FUNCTION_BLOCK FB_Symulacja IMPLEMENTS ITF_StanMaszyny
VAR_INPUT
	stParametry								: DUT_Symulacja_Parametry;
	stStanyPodzespolow						: DUT_Krajalnica_StanyPodzespolow;
	eTrybPracy								: E_PMLUnitMode;
END_VAR
VAR_OUTPUT
	//wyjscia zadziałania czujnikow 
	bCiecie1_Poczatek						: BOOL;
	bCiecie1_Koniec							: BOOL;
	bCiecie2_Poczatek						: BOOL;
	bCiecie2_Koniec							: BOOL;
	bPodawanieZabierakPoczatek				: BOOL;
	bPodawanieZabierakKoniec				: BOOL;
	bPodawaniePrzesuwaniePoczatek			: BOOL;
	bPodawaniePrzesuwanieKoniec				: BOOL;
	bCzujnikWaflaDoPodania					: BOOL;
	bCzujnikWaflaDoCiecia1					: BOOL;
	bCzujnikWaflaDoCiecia2					: BOOL;
END_VAR
VAR
	tonCiecie1_BazowanieCzasNaPowrot				: TON;           
	tonCiecie1_CiecieCzasNaCiecie					: TON;
	tonCiecie1_CiecieCzasNaPowrot					: TON;
	tonCiecie2_BazowanieCzasNaPowrot				: TON;
	tonCiecie2_CiecieCzasNaCiecie					: TON;
	tonCiecie2_CiecieCzasNaPowrot					: TON;
	tonPodawanieZabierak_BazowanieCzasNaPowrot		: TON;
	tonPodawaniePrzesuwanie_BazowanieCzasNaPowrot	: TON;
	tonPodawanieZabierak_PodawanieCzasNaPrace	: TON;
	tonPodawanieZabierak_PodawanieCzasNaPowrot		: TON;
	tonPodawaniePrzesuwanie_PodawanieCzasNaPobranie	: TON;
	tonPodawaniePrzesuwanie_PodawanieCzasNaPodanie	: TON;	
END_VAR

tonCiecie1_BazowanieCzasNaPowrot				(IN := stStanyPodzespolow.bCiecie1_Bazowanie ,
													PT := REAL_TO_TIME (stParametry.rCiecie1_BazowanieCzasNaPowrot));
tonCiecie1_CiecieCzasNaCiecie					(IN := stStanyPodzespolow.bCiecie1_Naped_WStroneKonca ,
													PT := REAL_TO_TIME (stParametry.rCiecie1_CiecieCzasNaPowrot));
tonCiecie1_CiecieCzasNaPowrot					(IN := stStanyPodzespolow.bCiecie1_Naped_WStronePoczatku ,
													PT := REAL_TO_TIME (stParametry.rCiecie1_CiecieCzasNaCiecie));

tonCiecie2_BazowanieCzasNaPowrot				(IN := stStanyPodzespolow.bCiecie2_Bazowanie ,
													PT := REAL_TO_TIME (stParametry.rCiecie2_BazowanieCzasNaPowrot));
tonCiecie2_CiecieCzasNaCiecie					(IN := stStanyPodzespolow.bCiecie2_Naped_WStroneKonca ,
													PT := REAL_TO_TIME (stParametry.rCiecie2_CiecieCzasNaPowrot));
tonCiecie2_CiecieCzasNaPowrot					(IN := stStanyPodzespolow.bCiecie2_Naped_WStronePoczatku ,
													PT := REAL_TO_TIME (stParametry.rCiecie2_CiecieCzasNaCiecie));

tonPodawanieZabierak_BazowanieCzasNaPowrot		(IN := stStanyPodzespolow.bPodawanie_Bazowanie AND 
														stStanyPodzespolow.bPodawanie_Zabierak_WStronePoczatku ,
													PT := REAL_TO_TIME (stParametry.rPodawanieZabierak_BazowanieCzasNaPowrot));
tonPodawaniePrzesuwanie_BazowanieCzasNaPowrot	(IN := stStanyPodzespolow.bPodawanie_Bazowanie AND 
														stStanyPodzespolow.bPodawanie_Przesuwanie_WStronePoczatku ,
													PT := REAL_TO_TIME (stParametry.rPodawanieZabierak_PodawanieCzasNaPowrot));
tonPodawanieZabierak_PodawanieCzasNaPrace		(IN := stStanyPodzespolow.bPodawanie_Podawanie AND
														stStanyPodzespolow.bPodawanie_zabierak_WStroneKonca ,
													PT := REAL_TO_TIME (stParametry.rPodawanieZabierak_PodawanieCzasNaPrace));
tonPodawanieZabierak_PodawanieCzasNaPowrot		(IN := stStanyPodzespolow.bPodawanie_Podawanie AND
														stStanyPodzespolow.bPodawanie_Zabierak_WStronePoczatku ,
													PT := REAL_TO_TIME (stParametry.rPodawaniePrzesuwanie_BazowanieCzasNaPowrot));
tonPodawaniePrzesuwanie_PodawanieCzasNaPobranie	(IN := stStanyPodzespolow.bPodawanie_Podawanie AND
														stStanyPodzespolow.bPodawanie_Przesuwanie_WStroneKonca ,
													PT := REAL_TO_TIME (stParametry.rPodawaniePrzesuwanie_PodawanieCzasNaPobranie));
tonPodawaniePrzesuwanie_PodawanieCzasNaPodanie	(IN := stStanyPodzespolow.bPodawanie_Podawanie AND
														stStanyPodzespolow.bPodawanie_Przesuwanie_WStronePoczatku ,
													PT := REAL_TO_TIME (stParametry.rPodawaniePrzesuwanie_PodawanieCzasNaPodanie));

(*==================================================================================================
								RJM Maszyny sp. z o.o.
									5.06.2022
	Stan maszyny Aborted - metoda pusta
 	v1.0	|| TC v 3.1.4024.29		|| - pierwsza wersja
==================================================================================================*)
METHOD SM_Aborted : BOOL
END_METHOD

(*==================================================================================================
								RJM Maszyny sp. z o.o.
									5.06.2022
	Stan maszyny Aborting - awaryjne zatrzymanie maszyny E-STOP
 	v1.0	|| TC v 3.1.4024.29		|| - pierwsza wersja
==================================================================================================*)
METHOD SM_Aborting : BOOL
SM_Aborting									:= TRUE;
END_METHOD

(*==================================================================================================
								RJM Maszyny sp. z o.o.
									5.06.2022
	Stan maszyny Clearing
 	v1.0	|| TC v 3.1.4024.29		|| - pierwsza wersja
==================================================================================================*)
METHOD SM_Clearing : BOOL
SM_Clearing									:= TRUE;
END_METHOD

(*==================================================================================================
								RJM Maszyny sp. z o.o.
									5.06.2022
	Stan maszyny Complete 
 	v1.0	|| TC v 3.1.4024.29		|| - pierwsza wersja
==================================================================================================*)
METHOD SM_Complete : BOOL
END_METHOD

(*==================================================================================================
								RJM Maszyny sp. z o.o.
									5.06.2022
	Stan maszyny Completing
 	v1.0	|| TC v 3.1.4024.29		|| - pierwsza wersja
==================================================================================================*)
METHOD SM_Completing : BOOL
END_METHOD

(*==================================================================================================
								RJM Maszyny sp. z o.o.
									5.06.2022
	Stan maszyny Execute
 	v1.0	|| TC v 3.1.4024.29		|| - pierwsza wersja
==================================================================================================*)
METHOD SM_Execute : BOOL
VAR_INPUT
	eTrybPracy	: E_PMLUnitMode;
END_VAR
END_METHOD

(*==================================================================================================
								RJM Maszyny sp. z o.o.
									5.06.2022
	Stan maszyny Held  - metoda pusta
 	v1.0	|| TC v 3.1.4024.29		|| - pierwsza wersja
==================================================================================================*)
METHOD SM_Held : BOOL
END_METHOD

(*==================================================================================================
								RJM Maszyny sp. z o.o.
									5.06.2022
	Stan maszyny Holding
 	v1.0	|| TC v 3.1.4024.29		|| - pierwsza wersja
==================================================================================================*)
METHOD SM_Holding : BOOL
END_METHOD

(*==================================================================================================
								RJM Maszyny sp. z o.o.
									5.06.2022
	Stan maszyny Idle
 	v1.0	|| TC v 3.1.4024.29		|| - pierwsza wersja
==================================================================================================*)
METHOD SM_Idle : BOOL
END_METHOD

(*==================================================================================================
								RJM Maszyny sp. z o.o.
									5.06.2022
	Stan maszyny Reseting - konczenie niedokocznonych cykli i powrot podzespolami do pozycji startowej
 	v1.0	|| TC v 3.1.4024.29		|| - pierwsza wersja
==================================================================================================*)
METHOD SM_Resetting : BOOL
VAR_INPUT
	eTrybPracy								: E_PMLUnitMode;
END_VAR
SM_Resetting								:= TRUE;
END_METHOD

(*==================================================================================================
								RJM Maszyny sp. z o.o.
									5.06.2022
	Stan maszyny Starting - Ustawienie elementów do pracy 
 	v1.0	|| TC v 3.1.4024.29		|| - pierwsza wersja
==================================================================================================*)
METHOD SM_Starting : BOOL
END_METHOD

(*==================================================================================================
								RJM Maszyny sp. z o.o.
									5.06.2022
	Stan maszyny Stoped - metoda pusta
 	v1.0	|| TC v 3.1.4024.29		|| - pierwsza wersja
==================================================================================================*)
METHOD SM_Stopped : BOOL
END_METHOD

(*==================================================================================================
								RJM Maszyny sp. z o.o.
									5.06.2022
	Stan maszyny Stopping - Zakonczenie aktualnych operacji nie zaczynamy kolejnych
 	v1.0	|| TC v 3.1.4024.29		|| - pierwsza wersja
==================================================================================================*)
METHOD SM_Stopping : BOOL
END_METHOD

(*==================================================================================================
								RJM Maszyny sp. z o.o.
									5.06.2022
	Stan maszyny Suspended - metoda pusta
 	v1.0	|| TC v 3.1.4024.29		|| - pierwsza wersja
==================================================================================================*)
METHOD SM_Suspended : BOOL
END_METHOD

(*==================================================================================================
								RJM Maszyny sp. z o.o.
									5.06.2022
	Stan maszyny Suspending
 	v1.0	|| TC v 3.1.4024.29		|| - pierwsza wersja
==================================================================================================*)
METHOD SM_Suspending : BOOL
END_METHOD

(*==================================================================================================
								RJM Maszyny sp. z o.o.
									5.06.2022
	Stan maszyny Unholding
 	v1.0	|| TC v 3.1.4024.29		|| - pierwsza wersja
==================================================================================================*)
METHOD SM_Unholding : BOOL
END_METHOD

(*==================================================================================================
								RJM Maszyny sp. z o.o.
									5.06.2022
	Stan maszyny Unsuspending
 	v1.0	|| TC v 3.1.4024.29		|| - pierwsza wersja
==================================================================================================*)
METHOD SM_Unsuspending : BOOL
END_METHOD

END_FUNCTION_BLOCK

(* stored: Version 1.1.0.1, ProductVersion 3.1.4024.11
   POU FB_Symulacja: Id {765dcd61-bc4a-4fd9-ac8e-50d6dcf33eec}, SpecialFunc None
   Method SM_Aborted: Id {9820e384-b0a1-4a66-b766-7943285c2ac4}
   Method SM_Aborting: Id {e9bc9ab0-0d62-45b3-87ed-c48facf26e6a}
   Method SM_Clearing: Id {d163b2b8-f211-4417-bbf5-77228b385af9}
   Method SM_Complete: Id {0f0e3d35-0984-42ea-aa82-088afcd7725d}
   Method SM_Completing: Id {09d9d436-b712-4447-9816-dcfd05c8572f}
   Method SM_Execute: Id {63969b11-f63c-4dbf-812a-15889dfbd297}
   Method SM_Held: Id {1322292e-a8f5-42f5-b961-fb202a5f24c3}
   Method SM_Holding: Id {01d50ea5-47c7-4cb4-8a36-ef46039a9500}
   Method SM_Idle: Id {ca33b034-1f43-4c44-8eac-87db46373658}
   Method SM_Resetting: Id {d2f071d2-07dd-4093-b4d5-b2873fa1fd86}
   Method SM_Starting: Id {cb29fb05-3558-4bc6-85d8-b4598b57210a}
   Method SM_Stopped: Id {e8c6cc90-3fea-4b85-b39c-66505ec65a00}
   Method SM_Stopping: Id {acf116d2-616d-4f22-b4b6-59579d770113}
   Method SM_Suspended: Id {103c2f79-faea-4685-a656-2e23f8e41503}
   Method SM_Suspending: Id {7ab1c70c-dd0f-4d06-b92d-790e6ad9975e}
   Method SM_Unholding: Id {e61b12f8-b1f2-4866-ba8e-9492f13e5f60}
   Method SM_Unsuspending: Id {8bd26fa7-7cca-4146-9c79-a16a802f7fde} *)
